{attribute addProperty BoxType "EJ7334-0008-0016"}
{attribute addProperty Id "EnableBIT10.1251ResetBIT10.1252"}
{attribute addProperty CRC "2531568008"}
{attribute addProperty SizeInBites "16"}
{attribute addProperty SizeInBytes "2"}
TYPE Control_96E4A988 :
STRUCT
	{attribute addProperty Name "Enable"}
	Enable : BOOL;
	{attribute addProperty Name "Reset"}
	Reset : BOOL;
	{attribute 'hide'}
	reserve_1_BIT_0 : BOOL;
	{attribute 'hide'}
	reserve_1_BIT_1 : BOOL;
	{attribute 'hide'}
	reserve_1_BIT_2 : BOOL;
	{attribute 'hide'}
	reserve_1_BIT_3 : BOOL;
	{attribute 'hide'}
	reserve_1_BIT_4 : BOOL;
	{attribute 'hide'}
	reserve_1_BIT_5 : BOOL;
	{attribute 'hide'}
	reserve_1_BIT_6 : BOOL;
	{attribute 'hide'}
	reserve_1_BIT_7 : BOOL;
	{attribute 'hide'}
	reserve_1_BIT_8 : BOOL;
	{attribute 'hide'}
	reserve_1_BIT_9 : BOOL;
	{attribute 'hide'}
	reserve_1_BIT_10 : BOOL;
	{attribute 'hide'}
	reserve_1_BIT_11 : BOOL;
	{attribute 'hide'}
	reserve_1_BIT_12 : BOOL;
	{attribute 'hide'}
	reserve_1_BIT_13 : BOOL;
END_STRUCT
END_TYPE

(* stored: Version 1.2.0.0, ProductVersion 3.1.4024.9
   DUT Control_96E4A988: Id {2e07f317-fccb-400c-8167-664f38804685} *)
